PROGRAM Mode
VAR
	fbMode       : FB_AutoManual;
   

    bAutoMode    : BOOL;
    bManualMode  : BOOL;
    bAutoReady   : BOOL;   // np. wyjście po opóźnieniu
END_VAR

fbMode(
    bControlOn  := bControlOn,
    bEstopOK    := bEstopOK,
    bMoveUp     := .bCylinderCmdUp,
    bMoveDown   := .bCylinderCmdDown,
    bCycleStart := .bCycleStartCmd,
    bCycleStop  := .bCycleStopCmd,
    tAutoDelay  := T#1S   // np. 1 sekunda opóźnienia
);

bAutoMode   := fbMode.bAutoMode;
bManualMode := fbMode.bManualMode;
bAutoReady  := fbMode.bAutoDelayed;


IF bAutoMode THEN
	GVL_HMI.sMode:='TRYB AUTOMATYCZNY';
	ELSE
		GVL_HMI.sMode:='TRYB RĘCZNY';	
END_IF

END_PROGRAM

(* stored: Version 1.1.0.1, ProductVersion 3.1.4024.15
   POU Mode: Id {76113f60-7519-4d83-8634-3c8589ca0881}, SpecialFunc None *)
